(* CODESYS project tcl_adsobjects.library
   Company: Red Rock Controls Limited
   Description: Unit Tests moved into library
   Version: 1.1.3.0
   Placeholder: tcl_AdsObjects
   Author: R Christopher
   Title: tcl_AdsObjects

Project tree, tasks and I/O mapping:
  libraries: Tc2_Standard, * (Beckhoff Automation GmbH); Tc2_System, * (Beckhoff Automation GmbH); Tc2_Utilities, * (Beckhoff Automation GmbH); Tc3_Module, * (Beckhoff Automation GmbH); tcl_BaseClasses, * (Red Rock Controls Limited); tcl_UnitTestLibrary, * (Red Rock Controls Limited)
  GVLs/
    global variables Constants
  POUs/
    Classes/
      By Index Group/
        function block T_AdsRead [ST]: Execute, Execution
        function block T_AdsReadWrite [ST]: Execute, Execution
        function block T_AdsWrite [ST]: Execute, Execution
      By Symbol Name/
        function block T_AdsReadBySymbolName [ST]: Execute, Execution
        function block T_AdsReadWriteBySymbolName [ST]: Execute, Execution
        function block T_AdsWriteBySymbolName [ST]: Execute, Execution
      On Change/
        StructureMonitor/
          function block T_StructureMonitor [ST]: Changed, Reset, Test
        function block T_AdsWriteOnChange [ST]: Execution, FB_exit, Initialise
  Tasks/
  UnitTests/
    Example/
      function block TInteger [ST]: Inc, Init
    program PB_TestRunner [ST]
    function block Test_ReadBySymbolName [ST]: FB_init
    function block Test_ReadBySymbolName_KeepingHandle [ST]: FB_init
    function block Test_ReadWriteBySymbolName [ST]: FB_init
    function block Test_ReadWriteBySymbolName_KeepingHandle [ST]: FB_init
    function block Test_WriteBySymbolName [ST]: FB_init
    function block Test_WriteBySymbolName_KeepingHandle [ST]: FB_init
  Version/
    global variables Global_Version
  text list GlobalTextList
*)

// GVLs/Constants
{attribute 'qualified_only'}
VAR_GLOBAL CONSTANT
    PortNo : UINT := 851;
END_VAR

// Version/Global_Version
{attribute 'TcGenerated'}
{attribute 'no-analysis'}
{attribute 'linkalways'}
// This function has been automatically generated from the project information.
VAR_GLOBAL CONSTANT
	{attribute 'const_non_replaced'}
	stLibVersion_tcl_AdsObjects : ST_LibVersion := (iMajor := 1, iMinor := 1, iBuild := 3, iRevision := 0, nFlags := 0, sVersion := '1.1.3.0');
END_VAR

// POUs/Classes/By Index Group/T_AdsRead
FUNCTION_BLOCK T_AdsRead
VAR
    _Execution : T_Execution;
    AdsRead1 : ADSREAD := (TMOUT := T#2S);
END_VAR

IF _Execution.Aborting THEN
    _Execution.SetAborted();
END_IF

AdsRead1(
	NETID:= , 
	PORT:= , 
	IDXGRP:= , 
	IDXOFFS:= , 
	LEN:= , 
	DESTADDR:= , 
	READ:= _Execution.Starting, 
	TMOUT:= , 
	BUSY=> , 
	ERR=> , 
	ERRID=> );

    
IF _Execution.Starting THEN
    _Execution.SetBusy();
END_IF
IF _Execution.Busy AND NOT AdsRead1.BUSY THEN
    IF AdsRead1.ERR THEN
        _Execution.SetError(F_ErrorIdToString(AdsRead1.ERRID));
    ELSE
        _Execution.SetDone();
	END_IF
END_IF

METHOD Execute : BOOL
VAR_INPUT
	AmsNetId:T_AmsNetid;
	Port:T_AmsPort;
	IndexGroup:UDINT; 
	IndexOffset:UDINT;
	DataLength:UDINT; 
	DataAddress:PVOID; 
END_VAR
AdsRead1.NETID      := AmsNetId;
AdsRead1.PORT       := Port;
AdsRead1.IDXGRP     := IndexGroup;
AdsRead1.IDXOFFS    := IndexOffset;
AdsRead1.LEN        := DataLength;
AdsRead1.DESTADDR   := DataAddress;

Execute := _Execution.Start();
END_METHOD

PROPERTY Execution : I_Execution
GET
Execution := _Execution;
END_GET
END_PROPERTY

END_FUNCTION_BLOCK

// POUs/Classes/By Index Group/T_AdsReadWrite
FUNCTION_BLOCK T_AdsReadWrite
VAR_INPUT
END_VAR
VAR_OUTPUT
END_VAR
VAR
    AdsReadWrite : ADSRDWRT;
    _Execution : T_Execution;
END_VAR

IF _Execution.Aborting THEN
    _Execution.SetAborted();
END_IF

AdsReadWrite(
	NETID:= , 
	PORT:= , 
	IDXGRP:= , 
	IDXOFFS:= , 
	WRITELEN:= , 
	READLEN:= , 
	SRCADDR:= , 
	DESTADDR:= , 
	WRTRD:= _Execution.Starting, 
	TMOUT:= , 
	BUSY=> , 
	ERR=> , 
	ERRID=> );
    
IF _Execution.Starting THEN
    _Execution.SetBusy();
END_IF
IF _Execution.Busy AND NOT AdsReadWrite.BUSY THEN
    IF AdsReadWrite.ERR THEN
        _Execution.SetError(F_ErrorIdToString(AdsReadWrite.ERRID));
    ELSE
        _Execution.SetDone();
	END_IF
END_IF

METHOD Execute : BOOL
VAR_INPUT
    AmsNetId             : T_AmsNetID;
    Port                 : T_AmsPort;
    IndexGroup           : UDINT;
    IndexOffset          : UDINT; 
    ArgsAddress          : PVOID; 
    ArgsLength           : UDINT; 
    ReturnValueAddress   : PVOID; 
    ReturnValueLength    : UDINT; 
END_VAR
IF _Execution.Start() THEN
    AdsReadWrite.NETID    := AmsNetId;
    AdsReadWrite.PORT     := Port;
    AdsReadWrite.IDXGRP   := IndexGroup;
    AdsReadWrite.IDXOFFS  := IndexOffset;
    // Data to be written...
    AdsReadWrite.SRCADDR  := ArgsAddress;
    AdsReadWrite.WRITELEN := ArgsLength;
    // Data returned...
    AdsReadWrite.DESTADDR := ReturnValueAddress;
    AdsReadWrite.READLEN  := ReturnValueLength;
END_IF
END_METHOD

PROPERTY Execution : I_Execution
GET
Execution := _Execution;
END_GET
END_PROPERTY

END_FUNCTION_BLOCK

// POUs/Classes/By Index Group/T_AdsWrite
FUNCTION_BLOCK T_AdsWrite
VAR
    _Execution : T_Execution;
    AdsWrite1 : ADSWRITE := (TMOUT := T#2S);
END_VAR

IF _Execution.Aborting THEN
    _Execution.SetAborted();
END_IF

AdsWrite1(
	NETID:= , 
	PORT:= , 
	IDXGRP:= , 
	IDXOFFS:= , 
	LEN:= , 
	SRCADDR:= , 
	WRITE:= _Execution.Starting, 
	TMOUT:= , 
	BUSY=> , 
	ERR=> , 
	ERRID=> );
    
IF _Execution.Starting THEN
    _Execution.SetBusy();
END_IF
IF _Execution.Busy AND NOT AdsWrite1.BUSY THEN
    IF AdsWrite1.ERR THEN
        _Execution.SetError(F_ErrorIdToString(AdsWrite1.ERRID));
    ELSE
        _Execution.SetDone();
	END_IF
END_IF

METHOD Execute : BOOL
VAR_INPUT
	AmsNetId:T_AmsNetid;
	Port:T_AmsPort;
	IndexGroup:UDINT; 
	IndexOffset:UDINT;
	DataLength:UDINT; 
	DataAddress:PVOID; 
END_VAR
AdsWrite1.NETID := AmsNetId;
AdsWrite1.PORT := Port;
AdsWrite1.IDXGRP := IndexGroup;
AdsWrite1.IDXOFFS := IndexOffset;
AdsWrite1.LEN := DataLength;
AdsWrite1.SRCADDR := DataAddress;
Execute := _Execution.Start();
END_METHOD

PROPERTY Execution : I_Execution
GET
Execution := _Execution;
END_GET
END_PROPERTY

END_FUNCTION_BLOCK

// POUs/Classes/By Symbol Name/T_AdsReadBySymbolName
FUNCTION_BLOCK T_AdsReadBySymbolName
VAR
    _Execution : T_Execution;
    StateMonitor : T_ValueMonitor;
    State : INT;

	AmsNetId : T_AmsNetId;
	Port : T_AmsPort;
	SymbolName : STRING;
    ReadDataAddress : PVOID;
    ReadDataLength : UDINT;
    KeepSymbolHandle    : BOOL;  
	SymbolHandle 	   :	DWORD := 0;
    RetryCounter : T_Counter;
    
    AdsReadWrite_GetSymHandle : T_AdsReadWrite;
    AdsRead_ReadFromSymbol : T_AdsRead;
    AdsWrite_ReleaseSymHandle : T_AdsWrite;
    
END_VAR
VAR CONSTANT
    sInit          : INT := 0;
    sGetHandle     : INT := 1;
    sReadData      : INT := 2;
    sReleaseHandle : INT := 3;
END_VAR

IF _Execution.Aborting THEN
    State := sInit;
    _Execution.SetAborted();
END_IF

StateMonitor.Test(State);
CASE State OF
    sInit:
        IF _Execution.Starting THEN
            _Execution.SetBusy();
            RetryCounter.Reset();
            IF SymbolHandle = 0 THEN
                State := sGetHandle;
            ELSE
                State := sReadData;
            END_IF
		END_IF
        
    sGetHandle:    
        IF StateMonitor.Changed THEN
            // Get a symbol handle from the runtime...
            AdsReadWrite_GetSymHandle.Execute(
                AmsNetId            := AmsNetId, 
                Port                := Port, 
                IndexGroup          := ADSIGRP_SYM_HNDBYNAME, 
                IndexOffset         := 0, 
                ArgsAddress         := ADR(SymbolName), 
                ArgsLength          := INT_TO_UDINT(LEN(SymbolName)), 
                ReturnValueAddress  := ADR(SymbolHandle), 
                ReturnValueLength   := SIZEOF(SymbolHandle));
        ELSE
            IF AdsReadWrite_GetSymHandle.Execution.Done THEN
                State := sReadData;
			END_IF
            IF AdsReadWrite_GetSymHandle.Execution.Error THEN
                _Execution.SetError(AdsReadWrite_GetSymHandle.Execution.ErrorMsg);
                SymbolHandle := 0;
                State := sInit;
			END_IF
        END_IF
        
    sReadData: 
        IF StateMonitor.Changed THEN
            // Read the data to from the symbol...
            AdsRead_ReadFromSymbol.Execute(
                AmsNetId        := AmsNetId, 
                Port            := Port, 
                IndexGroup      := ADSIGRP_SYM_VALBYHND, 
                IndexOffset     := SymbolHandle, 
                DataLength      := ReadDataLength, 
                DataAddress     := ReadDataAddress);
        ELSE
            IF AdsRead_ReadFromSymbol.Execution.Done THEN
                IF KeepSymbolHandle THEN
                    _Execution.SetDone();
                    State := sInit;
                ELSE
                    State := sReleaseHandle;
				END_IF

            ELSIF AdsRead_ReadFromSymbol.Execution.Error THEN
                // Retry if it failed due to an online change invalidating the symbol handle...
				IF RetryCounter.Value = 0 THEN
					RetryCounter.Inc();
					SymbolHandle := 0;
					State := sGetHandle;
				ELSE
					_Execution.SetError(AdsRead_ReadFromSymbol.Execution.ErrorMsg);
					SymbolHandle := 0;
					State := sInit;
				END_IF
			END_IF
		END_IF
            
     sReleaseHandle:    
        IF StateMonitor.Changed THEN
            // Release the symbol handle......
            AdsWrite_ReleaseSymHandle.Execute(
                AmsNetId        := AmsNetId, 
                Port            := Port, 
                IndexGroup      := ADSIGRP_SYM_RELEASEHND, 
                IndexOffset     := SymbolHandle, 
                DataLength      := 0, 
                DataAddress     := 0);
        ELSE
            IF AdsWrite_ReleaseSymHandle.Execution.Done THEN
                // Handle write error to the symbol...
                IF AdsRead_ReadFromSymbol.Execution.Error THEN
                    _Execution.SetError(AdsRead_ReadFromSymbol.Execution.ErrorMsg);
                ELSE
                    _Execution.SetDone();
				END_IF
                SymbolHandle := 0;
                State := sInit;
            ELSIF AdsWrite_ReleaseSymHandle.Execution.Error THEN
                // Handle release handle error...
                _Execution.SetError(AdsWrite_ReleaseSymHandle.Execution.ErrorMsg);
                SymbolHandle := 0;
                State := sInit;
			END_IF
		END_IF

END_CASE

AdsReadWrite_GetSymHandle();
AdsRead_ReadFromSymbol();
AdsWrite_ReleaseSymHandle();

METHOD Execute : BOOL
VAR_INPUT
	AmsNetId : T_AmsNetId;
	Port : T_AmsPort;
	SymbolName : STRING;
    ReadDataAddress : PVOID;
    ReadDataLength : UDINT;
    KeepSymbolHandle    : BOOL;  
END_VAR
THIS^.AmsNetId          := AmsNetId;
THIS^.Port              := Port;
THIS^.SymbolName        := SymbolName;
THIS^.ReadDataAddress   := ReadDataAddress;
THIS^.ReadDataLength    := ReadDataLength;
THIS^.KeepSymbolHandle  := KeepSymbolHandle;

Execute := _Execution.Start();
END_METHOD

PROPERTY Execution : I_Execution
GET
Execution := _Execution;
END_GET
END_PROPERTY

END_FUNCTION_BLOCK

// POUs/Classes/By Symbol Name/T_AdsReadWriteBySymbolName
FUNCTION_BLOCK T_AdsReadWriteBySymbolName
VAR
    _Execution          : T_Execution;
    StateMonitor        : T_ValueMonitor;
    State               : INT;
                        
	AmsNetId            : T_AmsNetId;
	Port                : T_AmsPort;
	SymbolName          : STRING;
    ReadDataAddress     : PVOID;
    ReadDataLength      : UDINT;
    WriteDataAddress    : PVOID;
    WriteDataLength     : UDINT;    
    KeepSymbolHandle    : BOOL;  
	SymbolHandle 	    :	DWORD := 0;
    RetryCounter        : T_Counter;
    
    AdsReadWrite_GetSymHandle : T_AdsReadWrite;
    AdsReadWrite_ToSymbol     : T_AdsReadWrite;
    AdsWrite_ReleaseSymHandle : T_AdsWrite;

END_VAR
VAR CONSTANT
    sInit          : INT := 0;
    sGetHandle     : INT := 1;
    sReadWrite     : INT := 2;
    sReleaseHandle : INT := 3;
END_VAR

IF _Execution.Aborting THEN
    State := sInit;
    _Execution.SetAborted();
END_IF

StateMonitor.Test(State);
CASE State OF
    sInit:
        IF _Execution.Starting THEN
            _Execution.SetBusy();
            RetryCounter.Reset();
            IF SymbolHandle = 0 THEN
                State := sGetHandle;
            ELSE
                State := sReadWrite;
            END_IF
		END_IF
        
    sGetHandle:    
        IF StateMonitor.Changed THEN
            // Get a symbol handle from the runtime...
            AdsReadWrite_GetSymHandle.Execute(
                AmsNetId            := AmsNetId, 
                Port                := Port, 
                IndexGroup          := ADSIGRP_SYM_HNDBYNAME, 
                IndexOffset         := 0, 
                ArgsAddress         := ADR(SymbolName), 
                ArgsLength          := INT_TO_UDINT(LEN(SymbolName)), 
                ReturnValueAddress  := ADR(SymbolHandle), 
                ReturnValueLength   := SIZEOF(SymbolHandle));
        ELSE
            IF AdsReadWrite_GetSymHandle.Execution.Done THEN
                State := sReadWrite;
			END_IF
            IF AdsReadWrite_GetSymHandle.Execution.Error THEN
                _Execution.SetError(AdsReadWrite_GetSymHandle.Execution.ErrorMsg);
                SymbolHandle := 0;
                State := sInit;
			END_IF
        END_IF
        
    sReadWrite:  
        IF StateMonitor.Changed THEN
            // Write the data to the symbol...
            AdsReadWrite_ToSymbol.Execute(
                AmsNetId           := AmsNetId, 
                Port               := Port, 
                IndexGroup         := ADSIGRP_SYM_VALBYHND, 
                IndexOffset        := SymbolHandle, 
                ArgsAddress        := WriteDataAddress, 
                ArgsLength         := WriteDataLength, 
                ReturnValueAddress := ReadDataAddress, 
                ReturnValueLength  := ReadDataLength);
            
        ELSE
            IF AdsReadWrite_ToSymbol.Execution.Done THEN
                IF KeepSymbolHandle THEN
                    _Execution.SetDone();
                    State := sInit;
                ELSE
                    State := sReleaseHandle;
				END_IF
                
            ELSIF AdsReadWrite_ToSymbol.Execution.Error THEN
                // Retry if it failed due to an online change invalidating the symbol handle...
				IF RetryCounter.Value = 0 THEN
					RetryCounter.Inc();
					SymbolHandle := 0;
					State := sGetHandle;
				ELSE
					_Execution.SetError(AdsReadWrite_ToSymbol.Execution.ErrorMsg);
					SymbolHandle := 0;
					State := sInit;
				END_IF
			END_IF
		END_IF

    sReleaseHandle:    
        IF StateMonitor.Changed THEN
            // Release the symbol handle......
            AdsWrite_ReleaseSymHandle.Execute(
                AmsNetId        := AmsNetId, 
                Port            := Port, 
                IndexGroup      := ADSIGRP_SYM_RELEASEHND, 
                IndexOffset     := SymbolHandle, 
                DataLength      := 0, 
                DataAddress     := 0);
        ELSE
            IF AdsWrite_ReleaseSymHandle.Execution.Done THEN
                // Handle write error to the symbol...
                IF AdsReadWrite_ToSymbol.Execution.Error THEN
                    _Execution.SetError(AdsReadWrite_ToSymbol.Execution.ErrorMsg);
                ELSE
                    _Execution.SetDone();
				END_IF
                SymbolHandle := 0;
                State := sInit;
            ELSIF AdsWrite_ReleaseSymHandle.Execution.Error THEN
                // Handle release handle error...
                _Execution.SetError(AdsWrite_ReleaseSymHandle.Execution.ErrorMsg);
                SymbolHandle := 0;
                State := sInit;
			END_IF
		END_IF

END_CASE

AdsReadWrite_GetSymHandle();
AdsReadWrite_ToSymbol();
AdsWrite_ReleaseSymHandle();

METHOD Execute : BOOL
VAR_INPUT
	AmsNetId : T_AmsNetId;
	Port : T_AmsPort;
	SymbolName : STRING;
    ReadDataAddress : PVOID;
    ReadDataLength : UDINT;
    WriteDataAddress : PVOID;
    WriteDataLength : UDINT;
    KeepSymbolHandle    : BOOL;  
END_VAR
THIS^.AmsNetId          := AmsNetId;
THIS^.Port              := Port;
THIS^.SymbolName        := SymbolName;
THIS^.ReadDataAddress   := ReadDataAddress;
THIS^.ReadDataLength    := ReadDataLength;
THIS^.WriteDataAddress  := WriteDataAddress;
THIS^.WriteDataLength   := WriteDataLength;
THIS^.KeepSymbolHandle  := KeepSymbolHandle;

Execute := _Execution.Start();
END_METHOD

PROPERTY Execution : I_Execution
GET
Execution := _Execution;
END_GET
END_PROPERTY

END_FUNCTION_BLOCK

// POUs/Classes/By Symbol Name/T_AdsWriteBySymbolName
FUNCTION_BLOCK T_AdsWriteBySymbolName
VAR
    _Execution : T_Execution;
    StateMonitor : T_ValueMonitor;
    State : INT;

	AmsNetId            : T_AmsNetId;
	Port                : T_AmsPort;
	SymbolName          : STRING;
    WriteDataAddress    : PVOID;
    WriteDataLength     : UDINT;    
    KeepSymbolHandle    : BOOL;  
	SymbolHandle 	    : DWORD := 0;
    RetryCounter        : T_Counter;

    AdsReadWrite_GetSymHandle : T_AdsReadWrite;
    AdsWrite_WriteToSymbol    : T_AdsWrite;
    AdsWrite_ReleaseSymHandle : T_AdsWrite;
END_VAR
VAR CONSTANT
    sInit          : INT := 0;
    sGetHandle     : INT := 1;
    sWriteData     : INT := 2;
    sReleaseHandle : INT := 3;
END_VAR

IF _Execution.Aborting THEN
    State := sInit;
    _Execution.SetAborted();
END_IF

StateMonitor.Test(State);
CASE State OF
    sInit:
        IF _Execution.Starting THEN
            _Execution.SetBusy();
            RetryCounter.Reset();
            IF SymbolHandle = 0 THEN
                State := sGetHandle;
            ELSE
                State := sWriteData;
            END_IF
		END_IF
        
    sGetHandle: 
        IF StateMonitor.Changed THEN
            // Get a symbol handle from the runtime...
            AdsReadWrite_GetSymHandle.Execute(
                AmsNetId            := AmsNetId, 
                Port                := Port, 
                IndexGroup          := ADSIGRP_SYM_HNDBYNAME, 
                IndexOffset         := 0, 
                ArgsAddress         := ADR(SymbolName), 
                ArgsLength          := INT_TO_UDINT(LEN(SymbolName)), 
                ReturnValueAddress  := ADR(SymbolHandle), 
                ReturnValueLength   := SIZEOF(SymbolHandle));
        ELSE
            IF AdsReadWrite_GetSymHandle.Execution.Done THEN
                State := sWriteData;
			END_IF
            IF AdsReadWrite_GetSymHandle.Execution.Error THEN
                _Execution.SetError(AdsReadWrite_GetSymHandle.Execution.ErrorMsg);
                SymbolHandle := 0;
                State := sInit;
			END_IF
        END_IF
        
    sWriteData: 
        IF StateMonitor.Changed THEN
            // Write the data to the symbol...
            AdsWrite_WriteToSymbol.Execute(
                AmsNetId        := AmsNetId, 
                Port            := Port, 
                IndexGroup      := ADSIGRP_SYM_VALBYHND, 
                IndexOffset     := SymbolHandle, 
                DataLength      := WriteDataLength, 
                DataAddress     := WriteDataAddress);
        ELSE
            IF AdsWrite_WriteToSymbol.Execution.Done THEN
                IF KeepSymbolHandle THEN
                    _Execution.SetDone();
                    State := sInit;
                ELSE
                    State := sReleaseHandle;
				END_IF
                
            ELSIF AdsWrite_WriteToSymbol.Execution.Error THEN
                // Retry if it failed due to an online change invalidating the symbol handle...
				IF RetryCounter.Value = 0 THEN
					RetryCounter.Inc();
					SymbolHandle := 0;
					State := sGetHandle;
				ELSE
					_Execution.SetError(AdsWrite_WriteToSymbol.Execution.ErrorMsg);
					SymbolHandle := 0;
					State := sInit;
				END_IF
			END_IF
		END_IF

    sReleaseHandle:    
        IF StateMonitor.Changed THEN
            // Release the symbol handle......
            AdsWrite_ReleaseSymHandle.Execute(
                AmsNetId        := AmsNetId, 
                Port            := Port, 
                IndexGroup      := ADSIGRP_SYM_RELEASEHND, 
                IndexOffset     := SymbolHandle, 
                DataLength      := 0, 
                DataAddress     := 0);
        ELSE
            IF AdsWrite_ReleaseSymHandle.Execution.Done THEN
                // Handle write error to the symbol...
                IF AdsWrite_WriteToSymbol.Execution.Error THEN
                    _Execution.SetError(AdsWrite_WriteToSymbol.Execution.ErrorMsg);
                ELSE
                    _Execution.SetDone();
				END_IF
                SymbolHandle := 0;
                State := sInit;
            ELSIF AdsWrite_ReleaseSymHandle.Execution.Error THEN
                // Handle release handle error...
                _Execution.SetError(AdsWrite_ReleaseSymHandle.Execution.ErrorMsg);
                SymbolHandle := 0;
                State := sInit;
            ELSIF AdsWrite_WriteToSymbol.Execution.Error THEN
                // Handle Write To Symbol error...
                _Execution.SetError(AdsWrite_WriteToSymbol.Execution.ErrorMsg);
                SymbolHandle := 0;
                State := sInit;
			END_IF
		END_IF

END_CASE

AdsReadWrite_GetSymHandle();
AdsWrite_WriteToSymbol();
AdsWrite_ReleaseSymHandle();

METHOD Execute : BOOL
VAR_INPUT
	AmsNetId            : T_AmsNetId;
	Port                : T_AmsPort;
	SymbolName          : STRING;
    WriteDataAddress    : PVOID;
    WriteDataLength     : UDINT;  
    KeepSymbolHandle    : BOOL;  
END_VAR
THIS^.AmsNetId          := AmsNetId;
THIS^.Port              := Port;
THIS^.SymbolName        := SymbolName;
THIS^.WriteDataAddress  := WriteDataAddress;
THIS^.WriteDataLength   := WriteDataLength;
THIS^.KeepSymbolHandle  := KeepSymbolHandle;

Execute := _Execution.Start();
END_METHOD

PROPERTY Execution : I_Execution
GET
Execution := _Execution;
END_GET
END_PROPERTY

END_FUNCTION_BLOCK

// POUs/Classes/On Change/StructureMonitor/T_StructureMonitor
{attribute 'no_explicit_call':= 'do not call this POU directly'}
FUNCTION_BLOCK T_StructureMonitor
VAR
    _Changed : BOOL;
    Stored_CRC : WORD := 16#FFFF;
END_VAR

PROPERTY Changed : BOOL
GET
Changed := _Changed;
END_GET
END_PROPERTY

METHOD Reset
VAR_INPUT
END_VAR
Stored_CRC := 16#FFFF;
END_METHOD

METHOD Test
VAR_INPUT
    StructureAddress : POINTER TO BYTE;
    StructureSize    : UDINT;
END_VAR
VAR
    CRC : WORD;
END_VAR
CRC := F_DATA_TO_CRC16_CCITT(
            pData:= StructureAddress, 
            cbData:= StructureSize, 
            crc:= 0);

_Changed := (CRC <> Stored_CRC);
    
IF Changed THEN
    Stored_CRC := CRC;
END_IF
END_METHOD

END_FUNCTION_BLOCK

// POUs/Classes/On Change/T_AdsWriteOnChange
FUNCTION_BLOCK T_AdsWriteOnChange
VAR
    DataAddress : PVOID;
    DataLength : UDINT;
    PollTime : LREAL; // seconds
    
    AmsNetId : T_AmsNetID;
    AmsPort : T_AmsPort;
    SymbolNameToWriteTo : T_Maxstring;
    
    StructureMonitor : T_StructureMonitor;
    ValueMonitor : T_ValueMonitorEx;
    OnTimer_Poll : T_OnTimer(PresetTime := 0.0);
    OnTimer_DisableOnError : T_OnTimer(PresetTime := 30.0);
    AdsWriteBySymbolName : T_AdsWriteBySymbolName;
    CommsError : BOOL;
    pBuffer : POINTER TO BYTE;
END_VAR

IF DataAddress = 0 OR DataLength = 0 OR pBuffer = 0 THEN
    RETURN;
END_IF

// Disable comms for 30s on comms error to avoid flooding ADS...
IF AdsWriteBySymbolName.Execution.Error THEN
    CommsError := TRUE;
END_IF

IF OnTimer_DisableOnError.Delay(CommsError) THEN
    CommsError := FALSE;
END_IF

// Poll timer:
IF OnTimer_Poll.Delay(AdsWriteBySymbolName.Execution.Ready AND NOT CommsError) THEN
    
    // Detect any change...
    StructureMonitor.Test(
        StructureAddress := DataAddress,
        StructureSize    := DataLength);
               
    // Write data...
    IF StructureMonitor.Changed THEN
        // Copy data to a buffer - it might have changed before we get round to sending it...
        MEMCPY(
            destAddr := pBuffer,
            srcAddr  := DataAddress,
            n        := DataLength);
            
        // send the data...    
        AdsWriteBySymbolName.Execute(
            AmsNetId         := AmsNetId, 
            Port             := AmsPort, 
            SymbolName       := SymbolNameToWriteTo, 
            WriteDataAddress := pBuffer,   
            WriteDataLength  := DataLength,
            KeepSymbolHandle := TRUE);
    END_IF
END_IF

AdsWriteBySymbolName();

PROPERTY Execution : I_Execution
GET
Execution := AdsWriteBySymbolName.Execution;
END_GET
END_PROPERTY

METHOD FB_exit : BOOL
VAR_INPUT
	bInCopyCode : BOOL; // if TRUE, the exit method is called for exiting an instance that is copied afterwards (online change).
END_VAR
IF NOT bInCopyCode THEN
    __DELETE(pBuffer);
END_IF
END_METHOD

METHOD Initialise
VAR_INPUT
    DataAddress : PVOID;
    DataLength : UDINT;
    PollTime : LREAL; // seconds
    
    AmsNetId : T_AmsNetID;
    AmsPort : T_AmsPort;
    SymbolNameToWriteTo : T_Maxstring;
END_VAR
THIS^.DataAddress         :=   DataAddress; 
THIS^.DataLength          :=   DataLength;
THIS^.PollTime            :=   PollTime; 

THIS^.AmsNetId            :=   AmsNetId;
THIS^.AmsPort             :=   AmsPort; 
THIS^.SymbolNameToWriteTo :=   SymbolNameToWriteTo; 

pBuffer := __NEW(BYTE,DataLength);
END_METHOD

END_FUNCTION_BLOCK

// UnitTests/Example/TInteger
{attribute 'hide'}
{attribute 'reflection'}
FUNCTION_BLOCK TInteger
VAR
    Value : INT;
END_VAR

{attribute 'TcRpcEnable'}
METHOD Inc : INT
VAR_INPUT
END_VAR
Value := Value + 1;
Inc := Value;
END_METHOD

METHOD Init
VAR_INPUT
    Value : INT;
END_VAR
THIS^.Value := Value;
END_METHOD

END_FUNCTION_BLOCK

// UnitTests/PB_TestRunner
PROGRAM PB_TestRunner
VAR
    Run : BOOL := TRUE;

    TestRunner : T_TestRunner('tcl_AdsObjects');
    
    Test_ReadBySymbolName                    : Test_ReadBySymbolName(AdsPort := _AppInfo.AdsPort);
    Test_ReadWriteBySymbolName               : Test_ReadWriteBySymbolName(AdsPort := _AppInfo.AdsPort);
    Test_WriteBySymbolName                   : Test_WriteBySymbolName(AdsPort := _AppInfo.AdsPort);
    Test_ReadBySymbolName_KeepingHandle      : Test_ReadBySymbolName_KeepingHandle(AdsPort := _AppInfo.AdsPort);
    Test_ReadWriteBySymbolName_KeepingHandle : Test_ReadWriteBySymbolName_KeepingHandle(AdsPort := _AppInfo.AdsPort);
    Test_WriteBySymbolName_KeepingHandle     : Test_WriteBySymbolName_KeepingHandle(AdsPort := _AppInfo.AdsPort);

END_VAR

IF Run THEN
    Run := FALSE;
    TestRunner.Initialise();
    TestRunner.AddTest(Test_ReadBySymbolName);
    TestRunner.AddTest(Test_ReadWriteBySymbolName);
    TestRunner.AddTest(Test_WriteBySymbolName);
    TestRunner.AddTest(Test_ReadBySymbolName_KeepingHandle);
    TestRunner.AddTest(Test_ReadWriteBySymbolName_KeepingHandle);
    TestRunner.AddTest(Test_WriteBySymbolName_KeepingHandle);
	TestRunner.Execute();
END_IF

TestRunner();

END_PROGRAM

// UnitTests/Test_ReadBySymbolName
FUNCTION_BLOCK Test_ReadBySymbolName EXTENDS T_UnitTestBase
VAR
    AdsReadBySymbolName : T_AdsReadBySymbolName;
    ValueToRead : INT;
    ReadResult  : INT;
    ScanCount : DINT;
	AdsPort : UINT;
END_VAR

CASE State OF
    0:
        ValueToRead := 1234;
        ReadResult  := 0;
        ScanCount   := 0;

        AdsReadBySymbolName.Execute(AmsNetId         := '',
                                    Port             := AdsPort,
                                    SymbolName       := 'PB_TestRunner.Test_ReadBySymbolName.ValueToRead',
                                    ReadDataAddress  := ADR(ReadResult),
                                    ReadDataLength   := SIZEOF(ReadResult),
                                    KeepSymbolHandle := FALSE);

        State := 10;

    10:
        ScanCount := ScanCount + 1;

        IF NOT AdsReadBySymbolName.Execution.Busy THEN
            State := 20;
        END_IF

    20:
        Assertion.AssertEquals_INT(Expected     := 1234,
                                   Actual       := ReadResult,
                                   Variablename := 'ReadResult');

        _TestResult.TestFailed    := Assertion.AssertionFailed;
        _TestResult.FailMessage   := Assertion._AssertionMessage;
        _TestResult.TestCompleted := TRUE;
        State                     := 0;
END_CASE

AdsReadBySymbolName();

METHOD FB_init : BOOL
VAR_INPUT
    bInitRetains : BOOL; // if TRUE, the retain variables are initialized (warm start / cold start)
    bInCopyCode  : BOOL; // if TRUE, the instance afterwards gets moved into the copy code (online change)
	AdsPort : UINT;
END_VAR
THIS^.AdsPort := AdsPort;
END_METHOD

END_FUNCTION_BLOCK

// UnitTests/Test_ReadWriteBySymbolName
FUNCTION_BLOCK Test_ReadWriteBySymbolName EXTENDS T_UnitTestBase
VAR
    AdsReadWriteBySymbolName : T_AdsReadWriteBySymbolName;
    TestInteger : TInteger;
    ReadWriteResult : INT;    
    ScanCount : DINT;
	AdsPort : UINT;
END_VAR

CASE State OF
    0:
        TestInteger.Init(1111);
        ReadWriteResult := 0;
        ScanCount       := 0;

        AdsReadWriteBySymbolName.Execute(AmsNetId         := '',
                                         Port             := AdsPort,
                                         SymbolName       := 'PB_TestRunner.Test_ReadWriteBySymbolName.TestInteger#Inc',
                                         ReadDataAddress  := ADR(ReadWriteResult),
                                         ReadDataLength   := SIZEOF(ReadWriteResult),
                                         WriteDataAddress := 0,
                                         WriteDataLength  := 0,
                                         KeepSymbolHandle := FALSE);

        State := 10;

    10:
        ScanCount := ScanCount + 1;

        IF NOT AdsReadWriteBySymbolName.Execution.Busy THEN
            State := 20;
        END_IF

    20:
        Assertion.AssertEquals_INT(Expected     := 1112,
                                   Actual       := ReadWriteResult,
                                   Variablename := 'ReadWriteResult');

        _TestResult.TestFailed    := Assertion.AssertionFailed;
        _TestResult.FailMessage   := Assertion._AssertionMessage;
        _TestResult.TestCompleted := TRUE;

        State := 0;
END_CASE

AdsReadWriteBySymbolName();

METHOD FB_init : BOOL
VAR_INPUT
    bInitRetains : BOOL; // if TRUE, the retain variables are initialized (warm start / cold start)
    bInCopyCode  : BOOL; // if TRUE, the instance afterwards gets moved into the copy code (online change)
	AdsPort : UINT;
END_VAR
THIS^.AdsPort := AdsPort;
END_METHOD

END_FUNCTION_BLOCK

// UnitTests/Test_WriteBySymbolName
FUNCTION_BLOCK Test_WriteBySymbolName EXTENDS T_UnitTestBase
VAR
    AdsWriteBySymbolName : T_AdsWriteBySymbolName;
    ValueToWrite : INT := 3456;
    WriteResult : INT;
    ScanCount : DINT;
	AdsPort : UINT;
END_VAR

CASE State OF
    0:
        ValueToWrite := 3456;
        WriteResult  := 0;
        ScanCount    := 0;

        AdsWriteBySymbolName.Execute(AmsNetId         := '',
                                     Port             := AdsPort,
                                     SymbolName       := 'PB_TestRunner.Test_WriteBySymbolName.WriteResult',
                                     WriteDataAddress := ADR(ValueToWrite),
                                     WriteDataLength  := SIZEOF(ValueToWrite),
                                     KeepSymbolHandle := FALSE);

        State := 10;

    10:
        ScanCount := ScanCount + 1;

        IF NOT AdsWriteBySymbolName.Execution.Busy THEN
            State := 20;
        END_IF

    20:
        Assertion.AssertEquals_INT(Expected     := 3456,
                                   Actual       := WriteResult,
                                   Variablename := 'WriteResult');

        _TestResult.TestFailed    := Assertion.AssertionFailed;
        _TestResult.FailMessage   := Assertion._AssertionMessage;
        _TestResult.TestCompleted := TRUE;

        State := 0;
END_CASE

AdsWriteBySymbolName();

METHOD FB_init : BOOL
VAR_INPUT
    bInitRetains : BOOL; // if TRUE, the retain variables are initialized (warm start / cold start)
    bInCopyCode  : BOOL; // if TRUE, the instance afterwards gets moved into the copy code (online change)
	AdsPort : UINT;
END_VAR
THIS^.AdsPort := AdsPort;
END_METHOD

END_FUNCTION_BLOCK

// UnitTests/Test_ReadBySymbolName_KeepingHandle
FUNCTION_BLOCK Test_ReadBySymbolName_KeepingHandle EXTENDS T_UnitTestBase
VAR
    AdsReadBySymbolName : T_AdsReadBySymbolName;
    ValueToRead : INT;
    ReadResult  : INT;
    ScanCount : DINT;
	AdsPort : UINT;
END_VAR

CASE State OF
    0:
        ValueToRead := 1234;
        ReadResult  := 0;
        ScanCount   := 0;

        AdsReadBySymbolName.Execute(AmsNetId         := '',
                                    Port             := AdsPort,
                                    SymbolName       := 'PB_TestRunner.Test_ReadBySymbolName_KeepingHandle.ValueToRead',
                                    ReadDataAddress  := ADR(ReadResult),
                                    ReadDataLength   := SIZEOF(ReadResult),
                                    KeepSymbolHandle := TRUE);

        State := 10;

    10:
        ScanCount := ScanCount + 1;

        IF NOT AdsReadBySymbolName.Execution.Busy THEN
            State := 20;
        END_IF

    20:
        Assertion.AssertEquals_INT(Expected     := 1234,
                                   Actual       := ReadResult,
                                   Variablename := 'ReadResult');

        _TestResult.TestFailed    := Assertion.AssertionFailed;
        _TestResult.FailMessage   := Assertion._AssertionMessage;
        _TestResult.TestCompleted := TRUE;

        State := 0;
END_CASE

AdsReadBySymbolName();

METHOD FB_init : BOOL
VAR_INPUT
    bInitRetains : BOOL; // if TRUE, the retain variables are initialized (warm start / cold start)
    bInCopyCode  : BOOL; // if TRUE, the instance afterwards gets moved into the copy code (online change)
	AdsPort : UINT;
END_VAR
THIS^.AdsPort := AdsPort;
END_METHOD

END_FUNCTION_BLOCK

// UnitTests/Test_ReadWriteBySymbolName_KeepingHandle
FUNCTION_BLOCK Test_ReadWriteBySymbolName_KeepingHandle EXTENDS T_UnitTestBase
VAR
    AdsReadWriteBySymbolName : T_AdsReadWriteBySymbolName;
    TestInteger : TInteger;
    ReadWriteResult : INT;    
    ScanCount : DINT;
	AdsPort : UINT;
END_VAR

CASE State OF
    0:
        TestInteger.Init(1111);
        ReadWriteResult := 0;
        ScanCount       := 0;

        AdsReadWriteBySymbolName.Execute(AmsNetId         := '',
                                         Port             := AdsPort,
                                         SymbolName       := 'PB_TestRunner.Test_ReadWriteBySymbolName_KeepingHandle.TestInteger#Inc',
                                         ReadDataAddress  := ADR(ReadWriteResult),
                                         ReadDataLength   := SIZEOF(ReadWriteResult),
                                         WriteDataAddress := 0,
                                         WriteDataLength  := 0,
                                         KeepSymbolHandle := TRUE);

        State := 10;

    10:
        ScanCount := ScanCount + 1;

        IF NOT AdsReadWriteBySymbolName.Execution.Busy THEN
            State := 20;
        END_IF

    20:
        Assertion.AssertEquals_INT(Expected     := 1112,
                                   Actual       := ReadWriteResult,
                                   Variablename := 'ReadWriteResult');

        _TestResult.TestFailed    := Assertion.AssertionFailed;
        _TestResult.FailMessage   := Assertion._AssertionMessage;
        _TestResult.TestCompleted := TRUE;

        State := 0;
END_CASE

AdsReadWriteBySymbolName();

METHOD FB_init : BOOL
VAR_INPUT
    bInitRetains : BOOL; // if TRUE, the retain variables are initialized (warm start / cold start)
    bInCopyCode  : BOOL; // if TRUE, the instance afterwards gets moved into the copy code (online change)
	AdsPort : UINT;
END_VAR
THIS^.AdsPort := AdsPort;
END_METHOD

END_FUNCTION_BLOCK

// UnitTests/Test_WriteBySymbolName_KeepingHandle
FUNCTION_BLOCK Test_WriteBySymbolName_KeepingHandle EXTENDS T_UnitTestBase
VAR
    AdsWriteBySymbolName : T_AdsWriteBySymbolName;
    ValueToWrite : INT := 3456;
    WriteResult : INT;
    ScanCount : DINT;
	AdsPort : UINT;
END_VAR

CASE State OF
    0:
        ValueToWrite := 3456;
        WriteResult  := 0;
        ScanCount    := 0;

        AdsWriteBySymbolName.Execute(AmsNetId         := '',
                                     Port             := AdsPort,
                                     SymbolName       := 'PB_TestRunner.Test_WriteBySymbolName_KeepingHandle.WriteResult',
                                     WriteDataAddress := ADR(ValueToWrite),
                                     WriteDataLength  := SIZEOF(ValueToWrite),
                                     KeepSymbolHandle := TRUE);

        State := 10;

    10:
        ScanCount := ScanCount + 1;

        IF NOT AdsWriteBySymbolName.Execution.Busy THEN
            State := 20;
        END_IF

    20:
        Assertion.AssertEquals_INT(Expected     := 3456,
                                   Actual       := WriteResult,
                                   Variablename := 'WriteResult');

        _TestResult.TestFailed    := Assertion.AssertionFailed;
        _TestResult.FailMessage   := Assertion._AssertionMessage;
        _TestResult.TestCompleted := TRUE;

        State := 0;
END_CASE

AdsWriteBySymbolName();

METHOD FB_init : BOOL
VAR_INPUT
    bInitRetains : BOOL; // if TRUE, the retain variables are initialized (warm start / cold start)
    bInCopyCode  : BOOL; // if TRUE, the instance afterwards gets moved into the copy code (online change)
	AdsPort : UINT;
END_VAR
THIS^.AdsPort := AdsPort;
END_METHOD

END_FUNCTION_BLOCK
